TYPE ST_HMI_DataSourceHistInfo : 
STRUCT
	sSPGuid: GUID;
	sAlyFilePath: STRING(255);
	sSourceType: STRING(80);
	sTopic: STRING(255);
	sLayoutID: GUID;
END_STRUCT
END_TYPE

(* stored: DUT ST_HMI_DataSourceHistInfo: Id 5fb18412-2726-45db-b3d8-a8fb4d3a2690 *)
